TYPE TcoUrRobotics_Status_v_1_x_x :
STRUCT
	ActionDescription : STRING(100);	
	State:TcoUrRobotics_State_v_1_x_x;



END_STRUCT
END_TYPE

(* stored: Version 1.1.0.1, ProductVersion 3.1.4024.12
   DUT TcoUrRobotics_Status_v_1_x_x: Id {e0165681-b349-01ba-02f1-bc7f8e208916} *)
